# EPICS StreamDevice protocol: src/keysight_B2900.proto
Terminator = LF;

getIDN {
    out "*IDN?";
    in "%\$1[^\n]";
    ExtraInput = Ignore;
}

# Generic

cmd {
    out "\$1";
}

getD {
    out "\$1?";
    in "%d";
    ExtraInput = Ignore;
}

setD {
    out "\$1 %d";
    @init {getD;}
}

getF {
    out "\$1?";
    in "%f";
    ExtraInput = Ignore;
}

setF {
    out "\$1 %f";
    @init {getF;}
}

getE {
    out "\$1?";
    in "%E";
    ExtraInput = Ignore;
}

setE {
    out "\$1 %E";
    @init {getE;}
}

getS {
    out "\$1?";
    in "%s";
    ExtraInput = Ignore;
}

setS {
    out "\$1 %s";
    @init {getS;}
}

getB {
    out "\$1?";
    in "%b";
    ExtraInput = Ignore;
}

setB {
    out "\$1 %b";
    @init {getB;}
}

getWF {
    out "\$2";
    in "%\$1[^\r\n]";
}

getArray {
    separator=",";
    out "\$1?";
    in "%f";
}

# Status and display command

# Trigger

# Delay

delay {
    out "DLAY %(\$1ChannelEdge)d,%(\$1ChannelLink)d,%e";
}

setDoutput {
    out "\$1 \$2,%d";
}

getDoutput {
    out "\$1?\$2";
    in "%d";
    ExtraInput = Ignore;
}

setDchannel {
    out "\$1 \$2,%d";
}

getDchannel {
    out "\$1?\$2";
    in "%d";
    ExtraInput = Ignore;
}

getDelay
{
    out "DLAY?\$2";
    in "%(\$1ChannelLink_RBV)d,%f";
    ExtraInput = Ignore;
}
